// TIA Portal V19 export
TYPE "C701_VAR_IF_LBS_TYPIC"
   STRUCT
      WRE { ExternalAccessible := 'False'; ExternalVisible := 'False'; ExternalWritable := 'False'} : USInt;   // Werkingsregime
      BMO_HAND { ExternalAccessible := 'False'; ExternalVisible := 'False'; ExternalWritable := 'False'} : Bool;   // TRUE = Werkingsregime is handmatig ingesteld via lokale bediening
      "Vrijgave pomp verwarmingsbat" { ExternalAccessible := 'False'; ExternalVisible := 'False'; ExternalWritable := 'False'} : Bool;   // Gaat naar if verwarmingskring CHECKEN OF DEZE POMP NU HIER INZIT OF IN DE KRING
      REQ_VE { ExternalAccessible := 'False'; ExternalVisible := 'False'; ExternalWritable := 'False'} : Bool;   // Warmtevraag voor kring verwarmingsbatterijen
      REQ_KO { ExternalAccessible := 'False'; ExternalVisible := 'False'; ExternalWritable := 'False'} : Bool;   // Koelvraag voor kring koelbatterijen (luchtgroep)
      STO { ExternalAccessible := 'False'; ExternalVisible := 'False'; ExternalWritable := 'False'} : Struct   // Opsomming van alle storingen
         A001 : Bool;   // Storing van de motorbeveiliging van pulsie ventilator
         A002 : Bool;   // Storing van de motorbeveiliging van extractie ventilator
         A003 : Bool;   // Fout drukmeting pulsie
         A004 : Bool;   // Fout drukmeting extractie
         A005 : Bool;   // Fout temperatuurmeting pulsie
         A006 : Bool;   // Fout temperatuurmeting extractie
         A007 : Bool;   // Fout temperatuurmeting buitenlucht
         A008 : Bool;   // Antivries alarm
         A009 : Bool;   // Filter vuil verse lucht
         A010 : Bool;   // Filter vuil extractie lucht
         AT01 : Bool;   // Foute terugmelding: damper verse lucht aangestuurd, terugmelding niet (of te laat) ontvangen
         AT02 : Bool;   // Foute terugmelding: damper extractie lucht aangestuurd, terugmelding niet (of te laat) ontvangen
         M001 : Bool;   // De pulsie ventilator is afgekoppeld via de werkschakelaar
         M002 : Bool;   // De extractie ventilator is afgekoppeld via de werkschakelaar
      END_STRUCT;
   END_STRUCT;
END_TYPE
